// TIA Portal V20 export
FUNCTION_BLOCK "FB_Fuel_Stand"   // FB1, FBD
{ S7_Optimized_Access := 'TRUE' }
// stored: SetENOAutomatically false
   VAR_INPUT
      iUnscaledMin : Real;
      iUnscaledMax : Real;
      iScaledMin : Real;
      iOffset : Real;
      iUnscaledAktVal : Int;
      iQuittieren : Bool;
      iImpuls : Bool;
      iStoerungUnterdr : Bool;
      iPipe_diameter : Bool;
      iMaxFlowRate : Real;
      iTemp_Raw : Word;
      Temp_Min : Real;
      Temp_Max : Real;
      Refrence_Temp : Real;
      iAssembly_Place : String;
   END_VAR
   VAR_OUTPUT
      outputfehler : "UDT_Flowmeter_Stoe";
   END_VAR
   VAR
      sFlowScaledValue : Real;
      eingang_80_plc : Bool;
      Buffer : Array[1..10] of Real;
      Index : DInt;
      Sum : Real;
      sScaledMax : Real;
      i : Int;
      sAvg : Real;
      bitte_schalte_an : Bool;
      sCyclecount : Real;
      IEC_Timer_0_Instance { S7_SetPoint := 'True'} : TON_TIME;
   END_VAR
   VAR_TEMP
      tVKE0 : Bool;
      tVKE1 : Bool;
      tdurchflussrate : Real;
      tbuffer01 : Int;
      tbuffer02 : Int;
      tbuffer03 : Int;
      tbuffer04 : DInt;
      tbuffer05 : Real;
      tbuffer06 : Word;
      tbuffer07 : Real;
      tNorm_FlowValue : Real;
      tNorm_TempValue : Real;
      "sensor-is-active" : Bool;
      tDrahtbruch : Bool;
   END_VAR
BEGIN

REGION Network 1
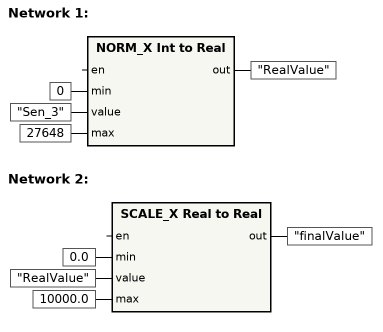
   "RealValue" := NORM_X(MIN := 0, VALUE := "Sen_3", MAX := 27648);
END_REGION

REGION Network 2
   "finalValue" := SCALE_X(MIN := 0.0, VALUE := "RealValue", MAX := 10000.0);
END_REGION
END_FUNCTION_BLOCK
